(* IEC 61131-3 sources: SIMERLIFT/logiwork_simerlift_80v/logiwork_simerlift_80v/HEMAbattery/src_FBD/fbdCommon/Library, 7 files *)

(* ---- DEMUX_4.iecfbd ---- *)
FUNCTION_BLOCK DEMUX_4
  {
    IN {index := 0};
    Select {index := 1};
    OUT_0 {index := 0};
    OUT_1 {index := 1};
    OUT_2 {index := 2};
    OUT_3 {index := 3};
    width := 200;
  }

  VAR_INPUT
    IN : UDINT := 0;
    Select : BYTE := 0;
  END_VAR
  VAR_OUTPUT
    OUT_1 : UDINT := 0;
    OUT_0 : UDINT := 0;
    OUT_2 : UDINT := 0;
    OUT_3 : UDINT := 0;
  END_VAR

  (*

    // Network 1:
    EQ(IN1 := Select, IN2 := 0, EQ => @C(11).EQ);
    SEL_UDINT(G := @C(11).EQ, IN0 := 0, IN1 := IN, SEL_UDINT => OUT_0);
    EQ(IN1 := Select, IN2 := 1, EQ => @C(14).EQ);
    SEL_UDINT(G := @C(14).EQ, IN0 := 0, IN1 := IN, SEL_UDINT => OUT_1);
    EQ(IN1 := Select, IN2 := 2, EQ => @C(18).EQ);
    SEL_UDINT(G := @C(18).EQ, IN0 := 0, IN1 := IN, SEL_UDINT => OUT_2);
    EQ(IN1 := Select, IN2 := 3, EQ => @C(21).EQ);
    SEL_UDINT(G := @C(21).EQ, IN0 := 0, IN1 := IN, SEL_UDINT => OUT_3);

  *)

  @C(42) : @F(SEL_UDINT), @R(590.0, 20.0, 120.0, 58.0), @I(@N(G), @L(9.5)), @I(@N(IN0), @L(29.5)), @I(@N(IN1), @L(49.5)), @O(@N(SEL_UDINT), @R(9.5));
  @C(48) : @F(SEL_UDINT), @R(590.0, 80.0, 120.0, 58.0), @I(@N(G), @L(9.5)), @I(@N(IN0), @L(29.5)), @I(@N(IN1), @L(49.5)), @O(@N(SEL_UDINT), @R(9.5));
  @C(54) : @F(SEL_UDINT), @R(590.0, 140.0, 120.0, 58.0), @I(@N(G), @L(9.5)), @I(@N(IN0), @L(29.5)), @I(@N(IN1), @L(49.5)), @O(@N(SEL_UDINT), @R(9.5));
  @C(53) : @F(SEL_UDINT), @R(590.0, 200.0, 120.0, 58.0), @I(@N(G), @L(9.5)), @I(@N(IN0), @L(29.5)), @I(@N(IN1), @L(49.5)), @O(@N(SEL_UDINT), @R(9.5));
  @C(11) : @F(EQ), @R(320.0, 20.0, 40.0, 38.0), BYTE, @I(@N(IN1), @L(9.5)), @I(@N(IN2), @L(29.5)), @O(@N(EQ), @R(9.5));
  @C(14) : @F(EQ), @R(320.0, 80.0, 40.0, 38.0), BYTE, @I(@N(IN1), @L(9.5)), @I(@N(IN2), @L(29.5)), @O(@N(EQ), @R(9.5));
  @C(18) : @F(EQ), @R(320.0, 140.0, 40.0, 38.0), BYTE, @I(@N(IN1), @L(9.5)), @I(@N(IN2), @L(29.5)), @O(@N(EQ), @R(9.5));
  @C(21) : @F(EQ), @R(320.0, 200.0, 40.0, 38.0), BYTE, @I(@N(IN1), @L(9.5)), @I(@N(IN2), @L(29.5)), @O(@N(EQ), @R(9.5));
  @VF(1) : @E(OUT_1), @R(750.0, 80.0, 220.0, 19.0);
  @VF(47) : @E(OUT_0), @R(750.0, 20.0, 220.0, 19.0);
  @VF(2) : @E(OUT_2), @R(750.0, 140.0, 220.0, 19.0);
  @VF(3) : @E(OUT_3), @R(750.0, 200.0, 220.0, 19.0);
  @VF(44) : @E(0), @R(440.0, 40.0, 110.0, 19.0), UDINT;
  @VF(50) : @E(0), @R(440.0, 100.0, 110.0, 19.0), UDINT;
  @VF(56) : @E(0), @R(440.0, 160.0, 110.0, 19.0), UDINT;
  @VF(58) : @E(0), @R(440.0, 220.0, 110.0, 19.0), UDINT;
  @VF(16) : @E(1), @R(130.0, 100.0, 110.0, 19.0), BYTE;
  @VF(19) : @E(2), @R(130.0, 160.0, 110.0, 19.0), BYTE;
  @VF(22) : @E(3), @R(130.0, 220.0, 110.0, 19.0), BYTE;
  @VF(185) : @E(0), @R(130.0, 40.0, 110.0, 19.0), BYTE;
  @VF(8) : @E(IN), @R(20.0, 60.0, 220.0, 19.0);
  @VF(9) : @E(Select), @R(20.0, 20.0, 220.0, 19.0);
  @CP(49) : 399.5, 69.5;
  @CP(51) : 399.5, 129.5;
  @CP(55) : 399.5, 189.5;
  @CP(57) : 399.5, 249.5;
  @CP(15) : 279.5, 29.5;
  @CP(36) : 279.5, 89.5;
  @CP(37) : 279.5, 149.5;
  @CP(38) : 279.5, 209.5;

  @G(10) :
     @L(@C(42).SEL_UDINT, @VF(47).i)
    ;
  @G(90) :
     @L(@C(48).SEL_UDINT, @VF(1).i)
    ;
  @G(91) :
     @L(@C(54).SEL_UDINT, @VF(2).i)
    ;
  @G(45) :
     @L(@VF(44).o, @C(42).IN0)
    ;
  @G(52) :
     @L(@VF(50).o, @C(48).IN0)
    ;
  @G(62) :
     @L(@VF(56).o, @C(54).IN0)
    ;
  @G(92) :
     @L(@C(53).SEL_UDINT, @VF(3).i)
    ;
  @G(60) :
     @L(@VF(58).o, @C(53).IN0)
    ;
  @G(46) :
     @L(@VF(8).o, @CP(49)),
     @L(@CP(49), @C(42).IN1),
     @L(@CP(49), @CP(51)),
     @L(@CP(51), @C(48).IN1),
     @L(@CP(51), @CP(55)),
     @L(@CP(55), @C(54).IN1),
     @L(@CP(55), @CP(57)),
     @L(@CP(57), @C(53).IN1)
    ;
  @G(43) :
     @L(@C(11).EQ, @C(42).G)
    ;
  @G(83) :
     @L(@C(14).EQ, @C(48).G)
    ;
  @G(84) :
     @L(@C(18).EQ, @C(54).G)
    ;
  @G(85) :
     @L(@C(21).EQ, @C(53).G)
    ;
  @G(12) :
     @L(@VF(9).o, @CP(15)),
     @L(@CP(15), @C(11).IN1),
     @L(@CP(15), @CP(36)),
     @L(@CP(36), @C(14).IN1),
     @L(@CP(36), @CP(37)),
     @L(@CP(37), @C(18).IN1),
     @L(@CP(37), @CP(38)),
     @L(@CP(38), @C(21).IN1)
    ;
  @G(13) :
     @L(@VF(185).o, @C(11).IN2)
    ;
  @G(17) :
     @L(@VF(16).o, @C(14).IN2)
    ;
  @G(20) :
     @L(@VF(19).o, @C(18).IN2)
    ;
  @G(23) :
     @L(@VF(22).o, @C(21).IN2)
    ;
END_FUNCTION_BLOCK

(* ---- Input_D.iecfbd ---- *)
FUNCTION_BLOCK Input_D
  {
    CH {index := 0};
    O {index := 0};
    width := 120;
    bgColor := "darkgray";
  }

  VAR
    ANLG1 : ANLG;
    Select_41 : Select_4;
  END_VAR
  VAR_INPUT
    CH : USINT := 0;
  END_VAR
  VAR_OUTPUT
    O : BYTE := 0;
  END_VAR

  (*

    // Network 1:
    ANLG1(ADC := TMSADC#A1, GRP := TMSADCGRP#G1, CH := CH);
    GE(IN1 := ANLG1.VAL, IN2 := 3000, GE => @C(5).GE);
    LE(IN1 := ANLG1.VAL, IN2 := 2100, LE => @C(6).LE);
    AND(IN1 := NOT @C(5).GE, IN2 := NOT @C(6).LE, AND => @C(24).AND);
    GE(IN1 := ANLG1.VAL, IN2 := 5000, GE => @C(34).GE);
    Select_41(In0 := 0, In1 := 1, In2 := 2, In3 := 3, S0 := @C(24).AND, S1 := @C(5).GE, S2 := @C(6).LE, S3 := @C(34).GE, i := 0);
    TO_BYTE(IN := Select_41.Q, TO_BYTE => O);

  *)

  @C(416) : @FB(ANLG1), @R(300.0, 120.0, 120.0, 58.0), @I(@N(ADC), @L(9.5)), @I(@N(GRP), @L(29.5)), @I(@N(CH), @L(49.5)), @O(@N(VAL), @R(9.5));
  @VF(417) : @E(TMSADC#A1), @R(40.0, 120.0, 220.0, 19.0);
  @VF(418) : @E(TMSADCGRP#G1), @R(40.0, 140.0, 220.0, 19.0);
  @VF(1) : @E(CH), @R(40.0, 160.0, 220.0, 19.0);
  @C(5) : @F(GE), @R(650.0, 120.0, 40.0, 38.0), UINT, @I(@N(IN1), @L(9.5)), @I(@N(IN2), @L(29.5)), @O(@N(GE), @R(9.5));
  @C(6) : @F(LE), @R(650.0, 160.0, 40.0, 38.0), UINT, @I(@N(IN1), @L(9.5)), @I(@N(IN2), @L(29.5)), @O(@N(LE), @R(9.5));
  @VF(447) : @E(3000), @R(500.0, 140.0, 110.0, 19.0), UINT;
  @VF(10) : @E(2100), @R(500.0, 180.0, 110.0, 19.0), UINT;
  @VF(15) : @E(2), @R(870.0, 180.0, 110.0, 19.0), WORD;
  @VF(17) : @E(1), @R(870.0, 140.0, 110.0, 19.0), WORD;
  @VF(19) : @E(0), @R(870.0, 100.0, 110.0, 19.0), WORD;
  @VF(22) : @E(0), @R(870.0, 260.0, 110.0, 19.0), WORD;
  @C(24) : @F(AND), @R(790.0, 80.0, 40.0, 38.0), BOOL, @I(@N(IN1), @L(9.5), @NEG), @I(@N(IN2), @L(29.5), @NEG), @O(@N(AND), @R(9.5));
  @VF(21) : @E(O), @R(1380.0, 80.0, 220.0, 19.0);
  @C(28) : @F(TO_BYTE), @R(1220.0, 80.0, 120.0, 18.0), WORD, @I(@N(IN), @L(9.5)), @O(@N(TO_BYTE), @R(9.5));
  @CF(376) : @R(0.0, 0.0, 240.0, 19.0), @T("DIGITAL INPUT");
  @CF(31) : @R(1380.0, 120.0, 220.0, 89.0), @T("OUTPUTS$N0 - Threshold$N1 - HS Input$N2 - LS Input$N3 - Fault");
  @VF(32) : @E(3), @R(870.0, 220.0, 110.0, 19.0), WORD;
  @C(34) : @F(GE), @R(650.0, 200.0, 40.0, 38.0), UINT, @I(@N(IN1), @L(9.5)), @I(@N(IN2), @L(29.5)), @O(@N(GE), @R(9.5));
  @VF(37) : @E(5000), @R(500.0, 220.0, 110.0, 19.0), UINT;
  @C(12) : @FB(Select_41), @R(1020.0, 80.0, 160.0, 198.0), @I(@N(In0), @L(29.5)), @I(@N(In1), @L(69.5)), @I(@N(In2), @L(109.5)), @I(@N(In3), @L(149.5)), @I(@N(S0), @L(9.5)), @I(@N(S1), @L(49.5)), @I(@N(S2), @L(89.5)), @I(@N(S3), @L(129.5)), @I(@N(i), @L(189.5)), @O(@N(Q), @R(9.5));
  @CP(8) : 459.5, 129.5;
  @CP(25) : 749.5, 169.5;
  @CP(26) : 729.5, 129.5;
  @CP(36) : 459.5, 169.5;

  @G(2) :
     @L(@VF(417).o, @C(416).ADC)
    ;
  @G(3) :
     @L(@VF(418).o, @C(416).GRP)
    ;
  @G(4) :
     @L(@VF(1).o, @C(416).CH)
    ;
  @G(7) :
     @L(@C(416).VAL, @CP(8)),
     @L(@CP(8), @C(5).IN1),
     @L(@CP(8), @CP(36)),
     @L(@CP(36), @C(6).IN1),
     @L(@CP(36), @C(34).IN1)
    ;
  @G(9) :
     @L(@VF(447).o, @C(5).IN2)
    ;
  @G(11) :
     @L(@VF(10).o, @C(6).IN2)
    ;
  @G(16) :
     @L(@VF(15).o, @C(12).In2)
    ;
  @G(18) :
     @L(@VF(17).o, @C(12).In1)
    ;
  @G(13) :
     @L(@C(5).GE, @CP(26)),
     @L(@CP(26), @C(24).IN1),
     @L(@CP(26), @C(12).S1)
    ;
  @G(14) :
     @L(@C(6).LE, @CP(25)),
     @L(@CP(25), @C(24).IN2),
     @L(@CP(25), @C(12).S2)
    ;
  @G(20) :
     @L(@VF(19).o, @C(12).In0)
    ;
  @G(23) :
     @L(@VF(22).o, @C(12).i)
    ;
  @G(27) :
     @L(@C(24).AND, @C(12).S0)
    ;
  @G(29) :
     @L(@C(12).Q, @C(28).IN)
    ;
  @G(30) :
     @L(@C(28).TO_BYTE, @VF(21).i)
    ;
  @G(33) :
     @L(@VF(32).o, @C(12).In3)
    ;
  @G(35) :
     @L(@C(34).GE, @C(12).S3)
    ;
  @G(38) :
     @L(@VF(37).o, @C(34).IN2)
    ;
END_FUNCTION_BLOCK

(* ---- Input_HS.iecfbd ---- *)
FUNCTION_BLOCK Input_HS
  {
    O {index := 0};
    CH {index := 0};
    bgColor := "darkgray";
    width := 120;
  }

  VAR
    ANLG1 : ANLG;
  END_VAR
  VAR_INPUT
    CH : USINT := 0;
  END_VAR
  VAR_OUTPUT
    O : BOOL := 0;
  END_VAR

  (*

    // Network 1:
    ANLG1(ADC := TMSADC#A1, GRP := TMSADCGRP#G2, CH := CH);
    GE(IN1 := ANLG1.VAL, IN2 := 3000, GE => O);

  *)

  @C(416) : @FB(ANLG1), @R(300.0, 40.0, 120.0, 58.0), @I(@N(ADC), @L(9.5)), @I(@N(GRP), @L(29.5)), @I(@N(CH), @L(49.5)), @O(@N(VAL), @R(9.5));
  @C(5) : @F(GE), @R(610.0, 40.0, 40.0, 38.0), UINT, @I(@N(IN1), @L(9.5)), @I(@N(IN2), @L(29.5)), @O(@N(GE), @R(9.5));
  @VF(1) : @E(CH), @R(40.0, 80.0, 220.0, 19.0);
  @VF(417) : @E(TMSADC#A1), @R(40.0, 40.0, 220.0, 19.0);
  @VF(418) : @E(TMSADCGRP#G2), @R(40.0, 60.0, 220.0, 19.0);
  @VF(447) : @E(3000), @R(460.0, 60.0, 110.0, 19.0), UINT;
  @VF(6) : @E(O), @R(690.0, 40.0, 220.0, 19.0);

  @G(2) :
     @L(@VF(417).o, @C(416).ADC)
    ;
  @G(3) :
     @L(@VF(418).o, @C(416).GRP)
    ;
  @G(4) :
     @L(@VF(1).o, @C(416).CH)
    ;
  @G(7) :
     @L(@C(416).VAL, @C(5).IN1)
    ;
  @G(9) :
     @L(@VF(447).o, @C(5).IN2)
    ;
  @G(8) :
     @L(@C(5).GE, @VF(6).i)
    ;
END_FUNCTION_BLOCK

(* ---- Input_LS.iecfbd ---- *)
FUNCTION_BLOCK Input_LS
  {
    CH {index := 0};
    O {index := 0};
    width := 120;
    bgColor := "darkgray";
  }

  VAR
    ANLG1 : ANLG;
  END_VAR
  VAR_INPUT
    CH : USINT := 0;
  END_VAR
  VAR_OUTPUT
    O : BOOL := 0;
  END_VAR

  (*

    // Network 1:
    ANLG1(ADC := TMSADC#A1, GRP := TMSADCGRP#G2, CH := CH);
    LE(IN1 := ANLG1.VAL, IN2 := 2230, LE => O);

  *)

  @C(416) : @FB(ANLG1), @R(300.0, 40.0, 120.0, 58.0), @I(@N(ADC), @L(9.5)), @I(@N(GRP), @L(29.5)), @I(@N(CH), @L(49.5)), @O(@N(VAL), @R(9.5));
  @C(6) : @F(LE), @R(610.0, 40.0, 40.0, 38.0), UINT, @I(@N(IN1), @L(9.5)), @I(@N(IN2), @L(29.5)), @O(@N(LE), @R(9.5));
  @VF(1) : @E(CH), @R(40.0, 80.0, 220.0, 19.0);
  @VF(417) : @E(TMSADC#A1), @R(40.0, 40.0, 220.0, 19.0);
  @VF(418) : @E(TMSADCGRP#G2), @R(40.0, 60.0, 220.0, 19.0);
  @VF(10) : @E(2230), @R(460.0, 60.0, 110.0, 19.0), UINT;
  @VF(5) : @E(O), @R(690.0, 40.0, 220.0, 19.0);

  @G(2) :
     @L(@VF(417).o, @C(416).ADC)
    ;
  @G(3) :
     @L(@VF(418).o, @C(416).GRP)
    ;
  @G(4) :
     @L(@VF(1).o, @C(416).CH)
    ;
  @G(7) :
     @L(@C(416).VAL, @C(6).IN1)
    ;
  @G(11) :
     @L(@VF(10).o, @C(6).IN2)
    ;
  @G(8) :
     @L(@C(6).LE, @VF(5).i)
    ;
END_FUNCTION_BLOCK

(* ---- Lineer_Function.iecfbd ---- *)
FUNCTION_BLOCK Lineer_Function
  {
    Y2 {index := 5};
    Y1 {index := 4};
    X2 {index := 2};
    X1 {index := 1};
    Error {loc := "right", index := 5};
    Input {index := 0};
    Output {index := 0};
    Lim_Output {index := 1};
    width := 200;
    height := 118;
  }

  VAR_INPUT
    Input : LREAL := 0;
    X1 : LREAL := 0;
    X2 : LREAL := 0;
    Y1 : LREAL := 0;
    Y2 : LREAL := 0;
  END_VAR
  VAR_OUTPUT
    Output : LREAL := 0;
    Error : BOOL := 0;
    Lim_Output : LREAL := 0;
  END_VAR

  (*

    // Network 1:
    SUB(IN1 := Y2, IN2 := Y1, SUB => @C(58).SUB);
    SUB(IN1 := X2, IN2 := X1, SUB => @C(59).SUB);
    DIV(IN1 := @C(58).SUB, IN2 := @C(59).SUB, DIV => @C(35).DIV);
    MUL(IN1 := X1, IN2 := @C(35).DIV, MUL => @C(60).MUL);
    SUB(IN1 := Y1, IN2 := @C(60).MUL, SUB => @C(61).SUB);
    MUL(IN1 := @C(35).DIV, IN2 := Input, MUL => @C(56).MUL);
    ADD(IN1 := @C(61).SUB, IN2 := @C(56).MUL, ADD => (@C(62).ADD, Output));
    LIMIT(MN := Y1, IN := @C(62).ADD, MX := Y2, LIMIT => Lim_Output);
    LE(IN1 := X2, IN2 := X1, LE => Error);

  *)

  @C(33) : @F(LIMIT), @R(990.0, 110.0, 120.0, 58.0), LREAL, @I(@N(MN), @L(9.5)), @I(@N(IN), @L(29.5)), @I(@N(MX), @L(49.5)), @O(@N(LIMIT), @R(9.5));
  @C(35) : @F(DIV), @R(440.0, 110.0, 40.0, 38.0), LREAL, @I(@N(IN1), @L(9.5)), @I(@N(IN2), @L(29.5)), @O(@N(DIV), @R(9.5));
  @C(56) : @F(MUL), @R(560.0, 170.0, 40.0, 38.0), LREAL, @I(@N(IN1), @L(9.5)), @I(@N(IN2), @L(29.5)), @O(@N(MUL), @R(9.5));
  @C(58) : @F(SUB), @R(360.0, 110.0, 40.0, 38.0), LREAL, @I(@N(IN1), @L(9.5)), @I(@N(IN2), @L(29.5)), @O(@N(SUB), @R(9.5));
  @C(59) : @F(SUB), @R(360.0, 150.0, 40.0, 38.0), LREAL, @I(@N(IN1), @L(9.5)), @I(@N(IN2), @L(29.5)), @O(@N(SUB), @R(9.5));
  @C(60) : @F(MUL), @R(560.0, 90.0, 40.0, 38.0), LREAL, @I(@N(IN1), @L(9.5)), @I(@N(IN2), @L(29.5)), @O(@N(MUL), @R(9.5));
  @C(61) : @F(SUB), @R(640.0, 70.0, 40.0, 38.0), LREAL, @I(@N(IN1), @L(9.5)), @I(@N(IN2), @L(29.5)), @O(@N(SUB), @R(9.5));
  @C(62) : @F(ADD), @R(720.0, 70.0, 40.0, 38.0), LREAL, @I(@N(IN1), @L(9.5)), @I(@N(IN2), @L(29.5)), @O(@N(ADD), @R(9.5));
  @VF(68) : @E(Y1), @R(840.0, 110.0, 110.0, 19.0);
  @VF(69) : @E(Lim_Output), @R(1150.0, 110.0, 220.0, 19.0);
  @VF(70) : @E(Y2), @R(840.0, 150.0, 110.0, 19.0);
  @VF(71) : @E(Output), @R(1150.0, 70.0, 220.0, 19.0);
  @VF(72) : @E(Input), @R(20.0, 190.0, 220.0, 19.0);
  @VF(73) : @E(X2), @R(20.0, 150.0, 220.0, 19.0);
  @VF(74) : @E(Y2), @R(20.0, 110.0, 220.0, 19.0);
  @VF(76) : @E(X1), @R(20.0, 90.0, 220.0, 19.0);
  @VF(77) : @E(Y1), @R(20.0, 70.0, 220.0, 19.0);
  @C(57) : @F(LE), @R(360.0, 210.0, 40.0, 38.0), LREAL, @I(@N(IN1), @L(9.5)), @I(@N(IN2), @L(29.5)), @O(@N(LE), @R(9.5));
  @VF(64) : @E(Error), @R(1150.0, 210.0, 220.0, 19.0);
  @CP(78) : 519.5, 119.5;
  @CP(79) : 799.5, 79.5;
  @CP(80) : 319.5, 79.5;
  @CP(81) : 299.5, 99.5;
  @CP(66) : 299.5, 179.5;
  @CP(2) : 319.5, 159.5;

  @G(87) :
     @L(@C(58).SUB, @C(35).IN1)
    ;
  @G(88) :
     @L(@C(59).SUB, @C(35).IN2)
    ;
  @G(89) :
     @L(@C(35).DIV, @CP(78)),
     @L(@CP(78), @C(60).IN2),
     @L(@CP(78), @C(56).IN1)
    ;
  @G(91) :
     @L(@VF(68).o, @C(33).MN)
    ;
  @G(92) :
     @L(@VF(70).o, @C(33).MX)
    ;
  @G(93) :
     @L(@C(33).LIMIT, @VF(69).i)
    ;
  @G(94) :
     @L(@CP(81), @C(60).IN1),
     @L(@CP(81), @CP(66)),
     @L(@VF(76).o, @CP(81)),
     @L(@CP(66), @C(59).IN2),
     @L(@CP(66), @C(57).IN2)
    ;
  @G(95) :
     @L(@C(60).MUL, @C(61).IN2)
    ;
  @G(96) :
     @L(@CP(80), @C(61).IN1),
     @L(@CP(80), @C(58).IN2),
     @L(@VF(77).o, @CP(80))
    ;
  @G(97) :
     @L(@C(62).ADD, @CP(79)),
     @L(@CP(79), @C(33).IN),
     @L(@CP(79), @VF(71).i)
    ;
  @G(98) :
     @L(@C(61).SUB, @C(62).IN1)
    ;
  @G(99) :
     @L(@C(56).MUL, @C(62).IN2)
    ;
  @G(100) :
     @L(@VF(73).o, @CP(2)),
     @L(@CP(2), @C(59).IN1),
     @L(@CP(2), @C(57).IN1)
    ;
  @G(102) :
     @L(@VF(72).o, @C(56).IN2)
    ;
  @G(65) :
     @L(@C(57).LE, @VF(64).i)
    ;
  @G(1) :
     @L(@VF(74).o, @C(58).IN1)
    ;
END_FUNCTION_BLOCK

(* ---- Select_2.iecfbd ---- *)
FUNCTION_BLOCK Select_2
  {
    In0 {index := 0};
    S0 {index := 1};
    In1 {index := 2};
    S1 {index := 3};
    i {index := 5};
    Q {index := 0};
  }

  VAR_INPUT
    In0 : WORD := 0;
    In1 : WORD := 0;
    S0 : BOOL := 0;
    S1 : BOOL := 0;
    i : BYTE := 0;
  END_VAR
  VAR_OUTPUT
    Q : WORD := 0;
  END_VAR

  (*

    // Network 1:
    SEL_WORD(G := S0, IN0 := i, IN1 := In0, SEL_WORD => @C(19).SEL_WORD);
    SEL_WORD(G := S1, IN0 := @C(19).SEL_WORD, IN1 := In1, SEL_WORD => Q);

  *)

  @C(22) : @F(SEL_WORD), @R(420.0, 40.0, 120.0, 58.0), @I(@N(G), @L(9.5)), @I(@N(IN0), @L(29.5)), @I(@N(IN1), @L(49.5)), @O(@N(SEL_WORD), @R(9.5));
  @C(19) : @F(SEL_WORD), @R(260.0, 100.0, 120.0, 58.0), @I(@N(G), @L(9.5)), @I(@N(IN0), @L(29.5)), @I(@N(IN1), @L(49.5)), @O(@N(SEL_WORD), @R(9.5));
  @VF(1) : @E(In0), @R(40.0, 140.0, 140.0, 19.0);
  @VF(2) : @E(In1), @R(40.0, 80.0, 140.0, 19.0);
  @VF(10) : @E(S1), @R(40.0, 40.0, 140.0, 19.0);
  @VF(17) : @E(i), @R(40.0, 120.0, 140.0, 19.0);
  @VF(9) : @E(S0), @R(40.0, 100.0, 140.0, 19.0);
  @VF(18) : @E(Q), @R(580.0, 40.0, 140.0, 19.0);

  @G(29) :
     @L(@VF(10).o, @C(22).G)
    ;
  @G(36) :
     @L(@VF(2).o, @C(22).IN1)
    ;
  @G(21) :
     @L(@VF(1).o, @C(19).IN1)
    ;
  @G(20) :
     @L(@VF(9).o, @C(19).G)
    ;
  @G(3) :
     @L(@VF(17).o, @C(19).IN0)
    ;
  @G(4) :
     @L(@C(19).SEL_WORD, @C(22).IN0)
    ;
  @G(5) :
     @L(@C(22).SEL_WORD, @VF(18).i)
    ;
END_FUNCTION_BLOCK

(* ---- Select_4.iecfbd ---- *)
FUNCTION_BLOCK Select_4
  {
    In0 {index := 1};
    In1 {index := 3};
    In2 {index := 5};
    In3 {index := 7};
    Q {index := 0};
    S0 {index := 0};
    S1 {index := 2};
    S2 {index := 4};
    S3 {index := 6};
    i {index := 9};
    width := 160;
    height := 198;
  }

  VAR_INPUT
    In0 : WORD := 0;
    In1 : WORD := 0;
    In2 : WORD := 0;
    In3 : WORD := 0;
    S0 : BOOL := 0;
    S1 : BOOL := 0;
    S2 : BOOL := 0;
    S3 : BOOL := 0;
    i : WORD := 0;
  END_VAR
  VAR_OUTPUT
    Q : WORD := 0;
  END_VAR

  (*

    // Network 1:
    SEL_WORD(G := S0, IN0 := i, IN1 := In0, SEL_WORD => @C(19).SEL_WORD);
    SEL_WORD(G := S1, IN0 := @C(19).SEL_WORD, IN1 := In1, SEL_WORD => @C(22).SEL_WORD);
    SEL_WORD(G := S2, IN0 := @C(22).SEL_WORD, IN1 := In2, SEL_WORD => @C(24).SEL_WORD);
    SEL_WORD(G := S3, IN0 := @C(24).SEL_WORD, IN1 := In3, SEL_WORD => Q);

  *)

  @C(19) : @F(SEL_WORD), @R(220.0, 220.0, 120.0, 58.0), @I(@N(G), @L(9.5)), @I(@N(IN0), @L(29.5)), @I(@N(IN1), @L(49.5)), @O(@N(SEL_WORD), @R(9.5));
  @C(22) : @F(SEL_WORD), @R(380.0, 160.0, 120.0, 58.0), @I(@N(G), @L(9.5)), @I(@N(IN0), @L(29.5)), @I(@N(IN1), @L(49.5)), @O(@N(SEL_WORD), @R(9.5));
  @C(24) : @F(SEL_WORD), @R(540.0, 100.0, 120.0, 58.0), @I(@N(G), @L(9.5)), @I(@N(IN0), @L(29.5)), @I(@N(IN1), @L(49.5)), @O(@N(SEL_WORD), @R(9.5));
  @C(26) : @F(SEL_WORD), @R(700.0, 40.0, 120.0, 58.0), @I(@N(G), @L(9.5)), @I(@N(IN0), @L(29.5)), @I(@N(IN1), @L(49.5)), @O(@N(SEL_WORD), @R(9.5));
  @VF(18) : @E(Q), @R(860.0, 40.0, 140.0, 19.0);
  @VF(1) : @E(In0), @R(40.0, 260.0, 140.0, 19.0);
  @VF(2) : @E(In1), @R(40.0, 200.0, 140.0, 19.0);
  @VF(3) : @E(In2), @R(40.0, 140.0, 140.0, 19.0);
  @VF(4) : @E(In3), @R(40.0, 80.0, 140.0, 19.0);
  @VF(9) : @E(S0), @R(40.0, 220.0, 140.0, 19.0);
  @VF(10) : @E(S1), @R(40.0, 160.0, 140.0, 19.0);
  @VF(11) : @E(S2), @R(40.0, 100.0, 140.0, 19.0);
  @VF(12) : @E(S3), @R(40.0, 40.0, 140.0, 19.0);
  @VF(17) : @E(i), @R(40.0, 240.0, 140.0, 19.0);

  @G(20) :
     @L(@VF(9).o, @C(19).G)
    ;
  @G(21) :
     @L(@VF(1).o, @C(19).IN1)
    ;
  @G(29) :
     @L(@VF(10).o, @C(22).G)
    ;
  @G(30) :
     @L(@VF(11).o, @C(24).G)
    ;
  @G(34) :
     @L(@VF(12).o, @C(26).G)
    ;
  @G(36) :
     @L(@VF(2).o, @C(22).IN1)
    ;
  @G(37) :
     @L(@VF(3).o, @C(24).IN1)
    ;
  @G(38) :
     @L(@VF(4).o, @C(26).IN1)
    ;
  @G(5) :
     @L(@C(26).SEL_WORD, @VF(18).i)
    ;
  @G(6) :
     @L(@VF(17).o, @C(19).IN0)
    ;
  @G(7) :
     @L(@C(24).SEL_WORD, @C(26).IN0)
    ;
  @G(8) :
     @L(@C(22).SEL_WORD, @C(24).IN0)
    ;
  @G(13) :
     @L(@C(19).SEL_WORD, @C(22).IN0)
    ;
END_FUNCTION_BLOCK
